FUNCTION_BLOCK OneDI
VAR_INPUT
	
	Value  :BOOL;
	Offline:BOOL;
	
END_VAR

VAR_TEMP
	i: INT;
	
END_VAR


i :=GVL.nInputCoilIndex;

GVL.mb_Input_Coils[i+0]:=Value;
GVL.mb_Input_Coils[i+1]:=Offline;

GVL.nInputCoilIndex:= i+2;

END_FUNCTION_BLOCK

(* stored: Version 1.1.0.1, ProductVersion 3.1.4024.12
   POU OneDI: Id {7826a84e-5769-45cc-bc21-f5bc3732cec9}, SpecialFunc None *)
